# B&R Automation Studio project NewPendant_NG4_11_05_25A
Automation Studio 4.9


## Configuration X20CP1585_MIG_HW_PS

### Task classes (Cpu.sw)
```
Cyclic#1 (cycle 800 us, tolerance 0 us):
  LincolnPS <- Universal.LincolnPS.prg
  Telnet <- Universal.Telnet.prg [disabled]
  TML_srv <- Universal.TML_srv.prg
  AVC_SYNCH <- FourAxisTigCtrl.AVC_SYNCH.prg
Cyclic#2 (cycle 2400 us, tolerance 24000 us):
  TIG_PSprc <- Universal.TIG_PSprc.prg
  WRST <- Universal.WRST.prg
  XMLHelper <- Universal.XMLHelper.prg
  BR_DC <- Universal.BR_DC.prg
  AVCprc <- Universal.AVCprc.prg
  OSC_TMLprc <- Universal.OSC_TMLprc.prg
  WIREprc <- Universal.WIREprc.prg
  HW_PSprc <- Universal.HW_PSprc.prg
  GasCoolPrc <- Universal.GasCoolPrc.prg
  WireBlkPrc <- Universal.WireBlkPrc.prg
  IndexPrc <- Universal.IndexPrc.prg
  TvlRotPrc <- Universal.TvlRotPrc.prg
Cyclic#3 (cycle 51200 us, tolerance 5120000 us):
  MV <- Universal.MV.prg
  HMI_M <- FourAxisTigCtrl.HMI_M.prg
  MiscOper <- Universal.MiscOper.prg
  PermSaving <- FourAxisTigCtrl.PermSaving.prg
  Main2 <- FourAxisTigCtrl.Main2.prg
  DC2DirMtr <- Universal.DC2DirMtr.prg
  TML_RLY <- Universal.TML_RLY.prg
Cyclic#5 (cycle 204800 us, tolerance 204800 us):
  HMI_Report <- FourAxisTigCtrl.HMI_Report.prg
Cyclic#8 (cycle 8000 us, tolerance 40000000 us):
  SuperMstr <- Universal.SuperMstr.prg
  FileOper <- Universal.FileOper.prg
  cJSONTest <- UDP.cJSON.cJSONTest.prg [disabled] (AdditionalLibraryDirectories=\Logical\UDP\sscanf2\, AdditionalLibraries=sscanf2-i386)
  udpserv <- UDP.paiUDPService.udpserv.prg [disabled]
  udpApp <- UDP.udpApp.prg [disabled]
  udpclient <- UDP.paiUDPService.udpclient.prg [disabled]
  udpsimonly <- UDP.udpsimonly.prg [disabled]
DataObjects: Acp10sys, PermObj_15, PermObj_16, PermObj_7, LogBook1, PermObj_3
VcDataObjects: Visu1 <- Visu1.dob, Visu2 <- Visu2.dob, Visu_M <- Visu_M.dob
Binaries: TCData, vccbtn, vcpdvnc, arialbd, vcmgr, vcgclass, vcfile, vccnum, vcfntttf, vcpkat, vcbclass, arial, visvc, vcalarm, vcdsloc, vctcal, vcpfx20, vccshape, vcshared, vcrt, vcnet, vcctext, vcdsint, vcpdsw, vccovl, vcchspot, Visu202, Visu201, udbdef, Visu203, vcpfar00, vcclbox, Visu_M02, vccbmp, Visu_M03, Visu_M01, arialbi, vccstr, vccline, vccddbox, vccpopup, Visu102, Visu101, Visu103, vccdt, Acp10map, acp10cfg, asfw, ashwd, arconfig, iomap, sysconf, ashwac
Libraries: bglibas, asstring, AsXml, sprintf2, AsUDP, Runtime, Acp10man, Acp10par, NcGlobal, sys_lib, brsystem, Library, dvframe, standard, fileio, asiotime, astime, dataobj, powerlnk, astcp, vcresman, visapi, ashw, asbrmath, ashydcon
```

### Hardware
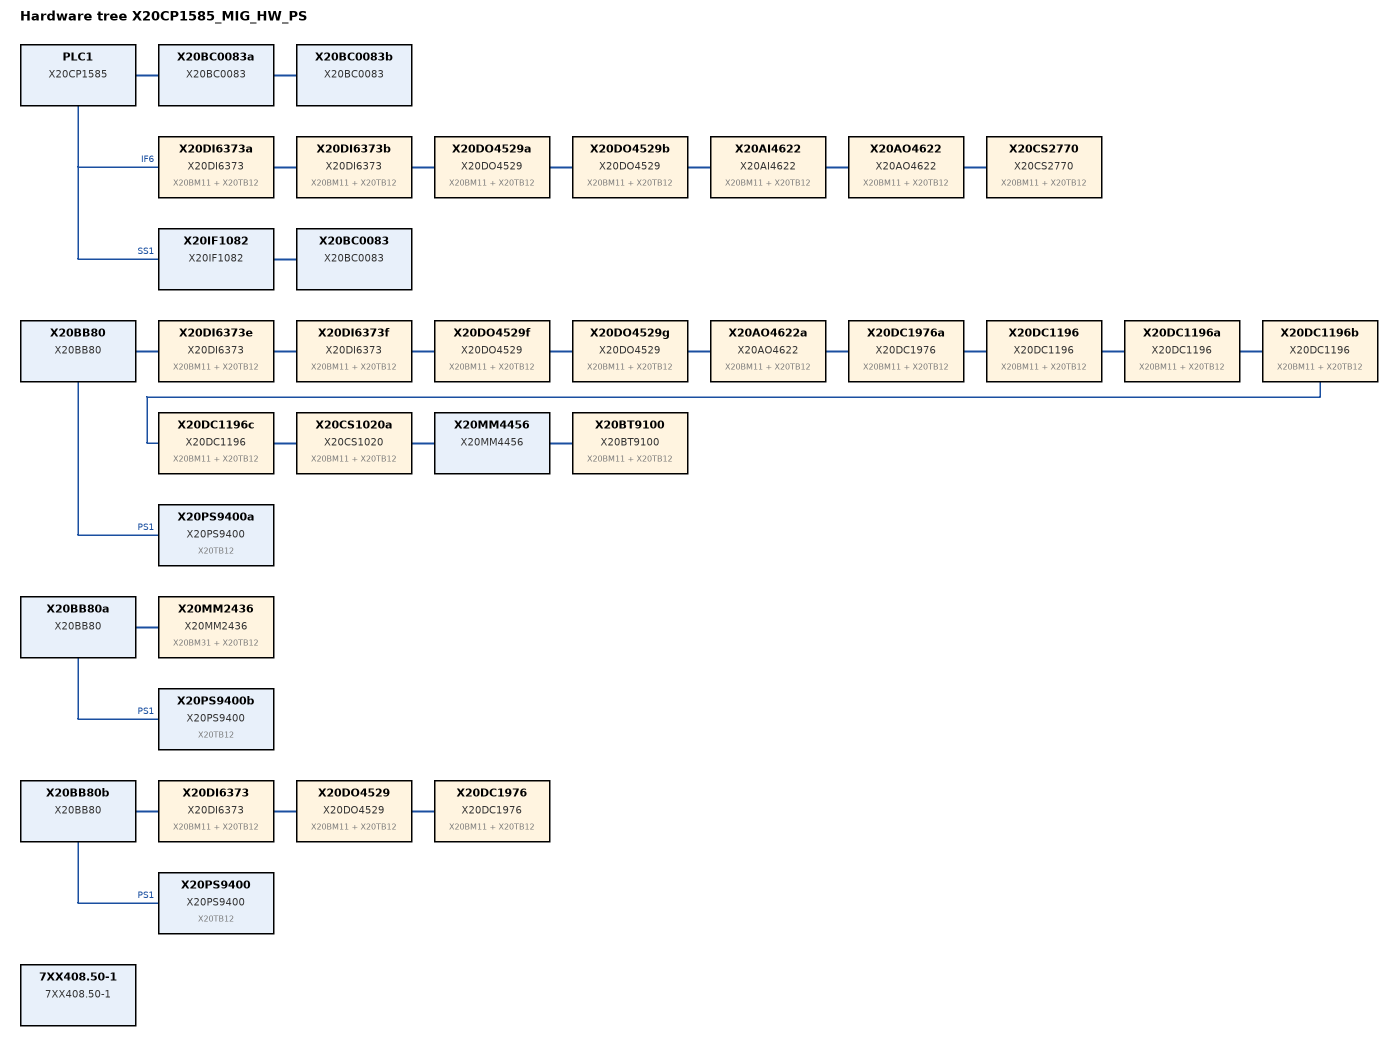
```
7XX408.50-1 : 7XX408.50-1 v1.2.0.0
  Supervision = off
  CounterMode = AB counter
PLC1 : X20CP1585 v1.10.0.0
  Connector IF2:
    ActivateDevice = 1
    Mode = Manual
    InternetAddress = 192.168.10.123
    SubnetMask = 255.255.255.0
    Vnc1
    VncVcObjectName1 = Visu_M
    VncKeyMappingFile1 = VC\PS2-Keyboard.dis
    VncMaxConnections1 = 3
    VncRefreshRate1 = 200
    VncTitle1 = Reports
    Vnc2
    VncVcObjectName2 = Visu2
    VncKeyMappingFile2 = VC\PS2-Keyboard1.dis
    VncPortNumber2 = 5901
    VncMaxConnections2 = 2
    VncRefreshRate2 = 100
    Vnc3
    VncVcObjectName3 = Visu1
    VncKeyMappingFile3 = VC\PS2-Keyboard14.dis
    VncPortNumber3 = 5902
    VncMaxConnections3 = 2
  Connector IF3:
    DNAConfiguration = manual
    CycleTime = 800
    EplNatSubnet = 192.168.102.0
    InaNodeNumber = 1
  Connector IF6:
    CycleTime = 800
  ConfigurationID = UnivCntrl-10-19-21F
  UserPartitionSize = 256
  UserRamSize = 770048
  PermanentPvSize = 96000
  RemanentGlobalPvSize = 15000
  VolatileGlobalPvSize = 3300000
  TimerDeviceType = EPLX2X
  TimerDevice = PLC1.IF3
  TaskClassIdleTime = 1600
  Cyclic1Duration = 800
  Cyclic1Tolerance = 0
  Cyclic1Stack = 16000
  Cyclic2Duration = 2400
  Cyclic2Tolerance = 24000
  Cyclic2Stack = 65536
  Cyclic3Duration = 51200
  Cyclic3Tolerance = 5120000
  Cyclic4Duration = 102400
  Cyclic4Tolerance = 102400
  Cyclic5Duration = 204800
  Cyclic5Tolerance = 204800
  Cyclic6Duration = 409600
  Cyclic6Tolerance = 409600
  Cyclic7Duration = 20000000
  Cyclic7Tolerance = 20000000
  Cyclic8Duration = 8000
  Cyclic8Tolerance = 40000000
  FileDevice1
  FileDeviceName1 = Data
  FileDevicePath1 = f:\Data
  FileDevice2
  FileDeviceName2 = WeldPrograms
  FileDevicePath2 = f:\WeldPrograms
  FileDevice3
  FileDeviceName3 = HMI
  FileDevicePath3 = f:\HMI
  FileDevice4
  FileDeviceName4 = CFG
  FileDevicePath4 = f:\CFG
  FileDevice5
  FileDeviceName5 = TEMP
  FileDevicePath5 = f:\TEMP
  FileDevice6
  FileDeviceName6 = REPORTS
  FileDevicePath6 = f:\Reports
  FtpUser1
  FtpUsername1 = anonymous
  FtpUserPassword1 = ilVrWe+rnGADVB+XCj+0qQ/lTsJeu4vW1xfWuH+9Xv8=
  FtpUserSalt1 = NATz6vdL
  FTPAccessRight1 = 0
X20AI4622 : X20AI4622 v1.2.0.0  [SS1 -> X20TB12c.SS; SL -> X20BM11c.SL1]
  Supervision = off
X20AO4622 : X20AO4622 v1.1.0.0  [SS1 -> X20TB12b.SS; SL -> X20BM11b.SL1]
  Supervision = off
X20AO4622a : X20AO4622 v1.1.0.0 (Disabled=true)  [SS1 -> X20TB12u.SS; SL -> X20BM11q.SL1]
  Supervision = off
X20BB80 : X20BB80 v1.0.2.0 (Disabled=true)
  Connector IF1 (Disabled=true)
    CycleTime = 800
X20BB80a : X20BB80 v1.0.2.0 (Disabled=true)
  Connector IF1 (Disabled=true)
    CycleTime = 800
    BusLength = 1
    Stations = 4
X20BB80b : X20BB80 v1.0.2.0 (Disabled=true)
  Connector IF1 (Disabled=true)
    CycleTime = 800
    AsyncPayload = 120
X20BC0083 : X20BC0083 v2.16.0.0 (Disabled=true)  [PLK1 -> X20IF1082.IF1 (NodeNumber=5) [Cable Type=PowerlinkCable, Length=10, Version=1.0.0.3]; SL -> X20BB80b.SL1]
  Supervision = off
X20BC0083a : X20BC0083 v2.16.0.0 (Disabled=true)  [PLK1 -> PLC1.IF3 (NodeNumber=6) [Cable Type=PowerlinkCable, Length=10, Version=1.0.0.3]; PLK2 -> X20BC0083b.PLK1 (NodeNumber=6) [Cable Type=PowerlinkCable, Length=10, Version=1.0.0.3]; SL -> X20BB80.SL1]
  Supervision = off
X20BC0083b : X20BC0083 v2.16.0.0 (Disabled=true)  [PLK1 -> X20BC0083a.PLK2 (NodeNumber=7) [Cable Type=PowerlinkCable, Length=10, Version=1.0.0.3]; SL -> X20BB80a.SL1]
  Supervision = off
X20BM11 : X20BM11 v1.1.0.0  [X2X1 -> X20BM11e.X2X2]
X20BM11a : X20BM11 v1.1.0.0  [X2X1 -> X20BM11d.X2X2]
X20BM11ab : X20BM11 v1.1.0.0 (Disabled=true)  [X2X1 -> X20BM11z.X2X2]
X20BM11b : X20BM11 v1.1.0.0  [X2X1 -> X20BM11c.X2X2]
X20BM11c : X20BM11 v1.1.0.0  [X2X1 -> X20BM11a.X2X2]
X20BM11d : X20BM11 v1.1.0.0  [X2X1 -> X20BM11.X2X2]
X20BM11e : X20BM11 v1.1.0.0  [X2X1 -> PLC1.IF6]
X20BM11l : X20BM11 v1.1.0.0  [X2X1 -> X20BM11b.X2X2]
X20BM11m : X20BM11 v1.1.0.0 (Disabled=true)  [X2X1 -> X20BB80.IF1]
X20BM11n : X20BM11 v1.1.0.0 (Disabled=true)  [X2X1 -> X20BM11m.X2X2]
X20BM11o : X20BM11 v1.1.0.0 (Disabled=true)  [X2X1 -> X20BM11n.X2X2]
X20BM11p : X20BM11 v1.1.0.0 (Disabled=true)  [X2X1 -> X20BM11o.X2X2]
X20BM11q : X20BM11 v1.1.0.0 (Disabled=true)  [X2X1 -> X20BM11p.X2X2]
X20BM11r : X20BM11 v1.1.0.0 (Disabled=true)  [X2X1 -> X20BM11q.X2X2]
X20BM11s : X20BM11 v1.1.0.0 (Disabled=true)  [X2X1 -> X20BM11r.X2X2]
X20BM11t : X20BM11 v1.1.0.0 (Disabled=true)  [X2X1 -> X20BM11s.X2X2]
X20BM11u : X20BM11 v1.1.0.0 (Disabled=true)  [X2X1 -> X20BM11t.X2X2]
X20BM11v : X20BM11 v1.1.0.0 (Disabled=true)  [X2X1 -> X20BM11u.X2X2]
X20BM11w : X20BM11 v1.1.0.0 (Disabled=true)  [X2X1 -> X20BM11v.X2X2]
X20BM11x : X20BM11 v1.1.0.0 (Disabled=true)  [X2X1 -> X20MM4456.X2X2]
X20BM11y : X20BM11 v1.1.0.0 (Disabled=true)  [X2X1 -> X20BB80b.IF1]
X20BM11z : X20BM11 v1.1.0.0 (Disabled=true)  [X2X1 -> X20BM11y.X2X2]
X20BM31 : X20BM31 v1.1.0.0 (Disabled=true)  [X2X1 -> X20BB80a.IF1]
X20BT9100 : X20BT9100 v1.3.0.0 (Disabled=true)  [SS1 -> X20TB12ab.SS; SL -> X20BM11x.SL1]
  Supervision = off
X20CS1020a : X20CS1020 v1.8.0.0 (Disabled=true)  [SS1 -> X20TB12aa.SS; SL -> X20BM11w.SL1]
  Connector IF1 (Disabled=true)
    ActivateIna = 0
  Supervision = off
X20CS2770 : X20CS2770 v1.9.1.0  [SS1 -> X20TB12n.SS; SL -> X20BM11l.SL1]
  Supervision = off
  CANdataFormat01 = UINT
  Baudrate02 = 250000
  CANdataFormat02 = UINT
X20DC1196 : X20DC1196 v1.4.0.0 (Disabled=true)  [SS1 -> X20TB12w.SS; SL -> X20BM11s.SL1]
  Supervision = off
X20DC1196a : X20DC1196 v1.4.0.0 (Disabled=true)  [SS1 -> X20TB12x.SS; SL -> X20BM11t.SL1]
  Supervision = off
X20DC1196b : X20DC1196 v1.4.0.0 (Disabled=true)  [SS1 -> X20TB12y.SS; SL -> X20BM11u.SL1]
  Supervision = off
X20DC1196c : X20DC1196 v1.4.0.0 (Disabled=true)  [SS1 -> X20TB12z.SS; SL -> X20BM11v.SL1]
  Supervision = off
X20DC1976 : X20DC1976 v1.3.0.0 (Disabled=true)  [SS1 -> X20TB12af.SS; SL -> X20BM11ab.SL1]
  Supervision = off
  BrokenWireConfig = off
X20DC1976a : X20DC1976 v1.3.0.0 (Disabled=true)  [SS1 -> X20TB12v.SS; SL -> X20BM11r.SL1]
  Supervision = off
  BrokenWireConfig = off
X20DI6373 : X20DI6373 v1.0.1.0 (Disabled=true)  [SS1 -> X20TB12ac.SS; SL -> X20BM11y.SL1]
  Supervision = off
X20DI6373a : X20DI6373 v1.0.1.0  [SS1 -> X20TB12e.SS; SL -> X20BM11e.SL1]
  Supervision = off
X20DI6373b : X20DI6373 v1.0.1.0  [SS1 -> X20TB12.SS; SL -> X20BM11.SL1]
  Supervision = off
X20DI6373e : X20DI6373 v1.0.1.0 (Disabled=true)  [SS1 -> X20TB12q.SS; SL -> X20BM11m.SL1]
  Supervision = off
X20DI6373f : X20DI6373 v1.0.1.0 (Disabled=true)  [SS1 -> X20TB12r.SS; SL -> X20BM11n.SL1]
  Supervision = off
X20DO4529 : X20DO4529 v1.2.0.0 (Disabled=true)  [SS1 -> X20TB12ad.SS; SL -> X20BM11z.SL1]
  Supervision = off
X20DO4529a : X20DO4529 v1.2.0.0  [SS1 -> X20TB12d.SS; SL -> X20BM11d.SL1]
  Supervision = off
X20DO4529b : X20DO4529 v1.2.0.0  [SS1 -> X20TB12a.SS; SL -> X20BM11a.SL1]
  Supervision = off
X20DO4529f : X20DO4529 v1.2.0.0 (Disabled=true)  [SS1 -> X20TB12s.SS; SL -> X20BM11o.SL1]
  Supervision = off
X20DO4529g : X20DO4529 v1.2.0.0 (Disabled=true)  [SS1 -> X20TB12t.SS; SL -> X20BM11p.SL1]
  Supervision = off
X20IF1082 : X20IF1082 v1.12.0.0 (Disabled=true)  [SS -> PLC1.SS1]
  Connector IF1 (Disabled=true)
    DNAConfiguration = manual
    CycleTime = 800
    InaNodeNumber = 1
X20MM2436 : X20MM2436 v1.6.0.0 (Disabled=true)  [SS1 -> X20TB12o.SS; SL -> X20BM31.SL1]
  Supervision = off
X20MM4456 : X20MM4456 v1.5.0.0 (Disabled=true)  [X2X1 -> X20BM11w.X2X2]
  Supervision = off
X20PS9400 : X20PS9400 v1.8.0.0 (Disabled=true)  [SS1 -> X20TB12ag.SS; PS -> X20BB80b.PS1]
  Supervision = off
  StatusInfo = off
X20PS9400a : X20PS9400 v1.8.0.0 (Disabled=true)  [SS1 -> X20TB12m.SS; PS -> X20BB80.PS1]
  Supervision = off
X20PS9400b : X20PS9400 v1.8.0.0 (Disabled=true)  [SS1 -> X20TB12p.SS; PS -> X20BB80a.PS1]
  Supervision = off
X20TB12 : X20TB12 v1.0.0.0
X20TB12a : X20TB12 v1.0.0.0
X20TB12aa : X20TB12 v1.0.0.0 (Disabled=true)
X20TB12ab : X20TB12 v1.0.0.0 (Disabled=true)
X20TB12ac : X20TB12 v1.0.0.0 (Disabled=true)
X20TB12ad : X20TB12 v1.0.0.0 (Disabled=true)
X20TB12af : X20TB12 v1.0.0.0 (Disabled=true)
X20TB12ag : X20TB12 v1.0.0.0 (Disabled=true)
X20TB12b : X20TB12 v1.0.0.0
X20TB12c : X20TB12 v1.0.0.0
X20TB12d : X20TB12 v1.0.0.0
X20TB12e : X20TB12 v1.0.0.0
X20TB12m : X20TB12 v1.0.0.0 (Disabled=true)
X20TB12n : X20TB12 v1.0.0.0
X20TB12o : X20TB12 v1.0.0.0 (Disabled=true)
X20TB12p : X20TB12 v1.0.0.0 (Disabled=true)
X20TB12q : X20TB12 v1.0.0.0 (Disabled=true)
X20TB12r : X20TB12 v1.0.0.0 (Disabled=true)
X20TB12s : X20TB12 v1.0.0.0 (Disabled=true)
X20TB12t : X20TB12 v1.0.0.0 (Disabled=true)
X20TB12u : X20TB12 v1.0.0.0 (Disabled=true)
X20TB12v : X20TB12 v1.0.0.0 (Disabled=true)
X20TB12w : X20TB12 v1.0.0.0 (Disabled=true)
X20TB12x : X20TB12 v1.0.0.0 (Disabled=true)
X20TB12y : X20TB12 v1.0.0.0 (Disabled=true)
X20TB12z : X20TB12 v1.0.0.0 (Disabled=true)
```

## Configuration X20CP1685_MIG_HW_PS

CPU X20CP1685, AutomationRuntime J4.93, Build 4.1.2, Safety 1.10, Vc V4.73.1

### IoMap.iom - PLC1/IoMap.iom
```iecst
(********************************************************************
 * COPYRIGHT -- wsi
 ********************************************************************
 * File: IoMap.iom
 * Author: wsi
 * Created: May 14, 2013
 ********************************************************************
 * IO mapping file
 ********************************************************************)
VAR_CONFIG
	::hardware.Inputs[0] AT %IX."X20DI6373e".DigitalInput01;
	::hardware.Inputs[1] AT %IX."X20DI6373e".DigitalInput02;
	::hardware.Inputs[2] AT %IX."X20DI6373e".DigitalInput03;
	::hardware.Inputs[3] AT %IX."X20DI6373e".DigitalInput04;
	::hardware.Inputs[4] AT %IX."X20DI6373e".DigitalInput05;
	::hardware.Inputs[6] AT %IX."X20DI6373f".DigitalInput01;
	::hardware.Inputs[7] AT %IX."X20DI6373f".DigitalInput02;
	::hardware.Inputs[8] AT %IX."X20DI6373f".DigitalInput03;
	::hardware.Inputs[9] AT %IX."X20DI6373f".DigitalInput04 INVERSE;
	Hardware[1].Inp[5] AT %IX."X20DI6373f".DigitalInput05; (*Gas Sensor*)
	Hardware[1].Inp[4] AT %IX."X20DI6373f".DigitalInput06; (*Coolant sensor*)
	::hardware.Inputs[13] AT %IX."X20DC1976a".DigitalInput02;
	::hardware.Inputs[14] AT %IX."X20DC1196".DigitalInput01;
	::hardware.Inputs[15] AT %IX."X20DC1196".DigitalInput02;
	::hardware.Inputs[16] AT %IX."X20DC1196a".DigitalInput01;
	::hardware.Inputs[17] AT %IX."X20DC1196a".DigitalInput02;
	::hardware.Inputs[18] AT %IX."X20DC1196b".DigitalInput01;
	::hardware.Inputs[19] AT %IX."X20DC1196b".DigitalInput02;
	::hardware.Inputs[20] AT %IX."X20DC1196c".DigitalInput01;
	::hardware.Inputs[21] AT %IX."X20DC1196c".DigitalInput02;
	::hardware.Outputs[0] AT %QX."X20DO4529f".DigitalOutput01;
	::hardware.Outputs[1] AT %QX."X20DO4529f".DigitalOutput02;
	::hardware.Outputs[2] AT %QX."X20DO4529f".DigitalOutput03;
	::hardware.Outputs[3] AT %QX."X20DO4529f".DigitalOutput04;
	::hardware.Outputs[4] AT %QX."X20DO4529g".DigitalOutput01;
	::hardware.Outputs[5] AT %QX."X20DO4529g".DigitalOutput02;
	::hardware.Outputs[6] AT %QX."X20DO4529g".DigitalOutput03;
	Hardware[1].Outp[4] AT %QX."X20DO4529g".DigitalOutput04; (*Gas Solenoid*)
	::hardware.AnalogOutputs[0] AT %QW."X20AO4622a".AnalogOutput01;
	::hardware.AnalogOutputs[1] AT %QW."X20AO4622a".AnalogOutput02;
	::hardware.AnalogOutputs[2] AT %QW."X20AO4622a".AnalogOutput03;
	::hardware.AnalogOutputs[3] AT %QW."X20AO4622a".AnalogOutput04;
	::motors[0].Hardware.PeriodDurationPWM AT %QW."X20MM4456".PeriodDurationPWM;
	::motors[0].Hardware.PulseWidthPWM AT %QW."X20MM4456".PulseWidthCurrentPWM01;
	::motors[1].Hardware.PulseWidthPWM AT %QW."X20MM4456".PulseWidthCurrentPWM02;
	::motors[2].Hardware.PulseWidthPWM AT %QW."X20MM4456".PulseWidthCurrentPWM03;
	::motors[3].Hardware.PulseWidthPWM AT %QW."X20MM4456".PulseWidthCurrentPWM04;
	::motors[0].Hardware.Counter AT %IW."X20DC1196".Encoder01;
	::motors[1].Hardware.Counter AT %IW."X20DC1196a".Encoder01;
	::motors[2].Hardware.Counter AT %IW."X20DC1196b".Encoder01;
	::motors[3].Hardware.Counter AT %IW."X20DC1196c".Encoder01;
	::hardware.Inputs[22] AT %IX."X20DI6373".DigitalInput01;
	::hardware.Inputs[23] AT %IX."X20DI6373".DigitalInput02;
	::hardware.Inputs[24] AT %IX."X20DI6373".DigitalInput03;
	::hardware.Inputs[25] AT %IX."X20DI6373".DigitalInput04;
	::hardware.Inputs[26] AT %IX."X20DI6373".DigitalInput05;
	::hardware.Inputs[27] AT %IX."X20DI6373".DigitalInput06;
	::hardware.Outputs[8] AT %QX."X20DO4529".DigitalOutput01;
	::hardware.Outputs[9] AT %QX."X20DO4529".DigitalOutput02;
	::hardware.Outputs[10] AT %QX."X20DO4529".DigitalOutput03;
	::hardware.Outputs[11] AT %QX."X20DO4529".DigitalOutput04;
	::hardware.Inputs[29] AT %IX."X20DC1976".DigitalInput02;
	::menu[1].Counter AT %IW."X20DC1976".Encoder01;
	::menu[1].MenuButton AT %IX."X20DC1976".DigitalInput01;
	::motors[0].Hardware.PWMError AT %IX."X20MM4456".PWMError01;
	::motors[0].Hardware.CurrentError AT %IX."X20MM4456".CurrentError01;
	::motors[0].Hardware.OverCurrentError AT %IX."X20MM4456".OverCurrentError01;
	::hardware.PWM_Status.UnderVoltageError AT %IX."X20MM4456".UnderVoltageError;
	::hardware.PWM_Status.VolatgeWarning AT %IX."X20MM4456".VoltageWarning;
	::hardware.PWM_Status.OverVoltageError AT %IX."X20MM4456".OverVoltageError;
	::hardware.PWM_Status.OvertempeatureError AT %IX."X20MM4456".OvertemperatureError;
	::motors[0].Hardware.ClearError AT %QX."X20MM4456".ResetCounter01;
	::motors[1].Hardware.ClearError AT %QX."X20MM4456".ClearError02;
	::motors[2].Hardware.ClearError AT %QX."X20MM4456".ClearError03;
	::motors[3].Hardware.ClearError AT %QX."X20MM4456".ClearError04;
	::motors[2].Hardware.PWMError AT %IX."X20MM4456".PWMError03;
	::motors[1].Hardware.PWMError AT %IX."X20MM4456".PWMError02;
	::motors[2].Hardware.CurrentError AT %IX."X20MM4456".CurrentError03;
	::motors[3].Hardware.CurrentError AT %IX."X20MM4456".CurrentError04;
	::motors[3].Hardware.PWMError AT %IX."X20MM4456".PWMError04;
	::motors[1].Hardware.OverCurrentError AT %IX."X20MM4456".OverCurrentError02;
	::motors[2].Hardware.OverCurrentError AT %IX."X20MM4456".OverCurrentError03;
	::motors[3].Hardware.OverCurrentError AT %IX."X20MM4456".OverCurrentError04;
	::motors[1].Hardware.CurrentError AT %IX."X20MM4456".CurrentError02;
	::Pendant[0].SerialNumber AT %ID."7XX408.50-1".SerialNumber;
	::Pendant[0].Inp[0] AT %IX."7XX408.50-1".DigitalInput03;
	::Pendant[0].Inp[1] AT %IX."7XX408.50-1".DigitalInput04;
	::Pendant[0].Inp[2] AT %IX."7XX408.50-1".DigitalInput05;
	::Pendant[0].Inp[3] AT %IX."7XX408.50-1".DigitalInput06;
	::Pendant[0].Inp[4] AT %IX."7XX408.50-1".DigitalInput07;
	::Pendant[0].Inp[5] AT %IX."7XX408.50-1".DigitalInput08;
	::Pendant[0].Inp[6] AT %IX."7XX408.50-1".DigitalInput09;
	::Pendant[0].Inp[7] AT %IX."7XX408.50-1".DigitalInput10;
	::Pendant[0].Inp[8] AT %IX."7XX408.50-1".DigitalInput11;
	::Pendant[0].Inp[9] AT %IX."7XX408.50-1".DigitalInput12;
	::Pendant[0].Inp[10] AT %IX."7XX408.50-1".DigitalInput13;
	::Pendant[0].Inp[11] AT %IX."7XX408.50-1".DigitalInput14;
	::Pendant[0].Inp[12] AT %IX."7XX408.50-1".DigitalInput15;
	::Pendant[0].Inp[13] AT %IX."7XX408.50-1".DigitalInput16;
	::Pendant[0].Outp[0] AT %QX."7XX408.50-1".DigitalOutput01;
	::Pendant[0].Outp[1] AT %QX."7XX408.50-1".DigitalOutput02;
	::Pendant[0].Outp[2] AT %QX."7XX408.50-1".DigitalOutput03;
	::Pendant[0].Outp[3] AT %QX."7XX408.50-1".DigitalOutput04;
	::Pendant[0].Outp[4] AT %QX."7XX408.50-1".DigitalOutput05;
	::Pendant[0].Outp[5] AT %QX."7XX408.50-1".DigitalOutput06;
	::Pendant[0].Outp[6] AT %QX."7XX408.50-1".DigitalOutput07;
	::Pendant[0].Outp[7] AT %QX."7XX408.50-1".DigitalOutput08;
	::Pendant[0].Outp[8] AT %QX."7XX408.50-1".DigitalOutput09;
	::Pendant[0].Outp[9] AT %QX."7XX408.50-1".DigitalOutput10;
	::Pendant[0].Outp[10] AT %QX."7XX408.50-1".DigitalOutput11;
	::Pendant[0].Outp[11] AT %QX."7XX408.50-1".DigitalOutput12;
	::Pendant[0].Outp[12] AT %QX."7XX408.50-1".DigitalOutput13;
	::Pendant[0].Outp[13] AT %QX."7XX408.50-1".DigitalOutput14;
	::Pendant[0].Outp[14] AT %QX."7XX408.50-1".DigitalOutput15;
	::Pendant[0].Outp[15] AT %QX."7XX408.50-1".DigitalOutput16;
	::Pendant[0].ABEncoder AT %ID."7XX408.50-1".ABEncoder01;
	::Pendant[0].NotWheelReset AT %QX."7XX408.50-1".NotCounterReset;
	::TML_mgr[0].hrdw[0].RXCount AT %IB."X20CS2770".RX01Count;
	::TML_mgr[0].hrdw[0].TXCountReadBack AT %IB."X20CS2770".TX01CountReadBack;
	::TML_mgr[0].hrdw[0].RXDataSize0 AT %IB."X20CS2770".RX01DataSize;
	::TML_mgr[0].hrdw[0].RXIdent0 AT %ID."X20CS2770".RX01Ident;
	::TML_mgr[0].hrdw[0].RXData0Word0[0] AT %IW."X20CS2770".RX01DataWord0;
	::TML_mgr[0].hrdw[0].RXData0Word0[1] AT %IW."X20CS2770".RX01DataWord1;
	::TML_mgr[0].hrdw[0].RXData0Word0[2] AT %IW."X20CS2770".RX01DataWord2;
	::TML_mgr[0].hrdw[0].RXData0Word0[3] AT %IW."X20CS2770".RX01DataWord3;
	::TML_mgr[0].hrdw[0].TXCount AT %QB."X20CS2770".TX01Count;
	::TML_mgr[0].hrdw[0].TXDataSize AT %QB."X20CS2770".TX01DataSize; (*Data length TX object *)
	::TML_mgr[0].hrdw[0].TXIdent AT %QD."X20CS2770".TX01Ident;
	::TML_mgr[0].hrdw[0].TXDataWord0[0] AT %QW."X20CS2770".TX01DataWord0;
	::TML_mgr[0].hrdw[0].TXDataWord0[1] AT %QW."X20CS2770".TX01DataWord1;
	::TML_mgr[0].hrdw[0].TXDataWord0[2] AT %QW."X20CS2770".TX01DataWord2;
	::TML_mgr[0].hrdw[0].TXDataWord0[3] AT %QW."X20CS2770".TX01DataWord3;
	::TML_mgr[0].hrdw[1].RXCount AT %IB."X20CS2770".RX02Count;
	::TML_mgr[0].hrdw[1].TXCountReadBack AT %IB."X20CS2770".TX02CountReadBack;
	::TML_mgr[0].hrdw[1].RXDataSize0 AT %IB."X20CS2770".RX02DataSize;
	::TML_mgr[0].hrdw[1].RXIdent0 AT %ID."X20CS2770".RX02Ident;
	::TML_mgr[0].hrdw[1].RXData0Word0[0] AT %IW."X20CS2770".RX02DataWord0;
	::TML_mgr[0].hrdw[1].RXData0Word0[1] AT %IW."X20CS2770".RX02DataWord1;
	::TML_mgr[0].hrdw[1].RXData0Word0[2] AT %IW."X20CS2770".RX02DataWord2;
	::TML_mgr[0].hrdw[1].RXData0Word0[3] AT %IW."X20CS2770".RX02DataWord3;
	::TML_mgr[0].hrdw[1].TXCount AT %QB."X20CS2770".TX02Count;
	::TML_mgr[0].hrdw[1].TXDataSize AT %QB."X20CS2770".TX02DataSize; (*Data length TX object *)
	::TML_mgr[0].hrdw[1].TXIdent AT %QD."X20CS2770".TX02Ident;
	::TML_mgr[0].hrdw[1].TXDataWord0[0] AT %QW."X20CS2770".TX02DataWord0;
	::TML_mgr[0].hrdw[1].TXDataWord0[1] AT %QW."X20CS2770".TX02DataWord1;
	::TML_mgr[0].hrdw[1].TXDataWord0[2] AT %QW."X20CS2770".TX02DataWord2;
	::TML_mgr[0].hrdw[1].TXDataWord0[3] AT %QW."X20CS2770".TX02DataWord3;
	::Hardware[2].PWM[0].PulseWidthPWM[0] AT %QW."X20MM2436".PulseWidthCurrentPWM01;
	::Hardware[2].PWM[0].PulseWidthPWM[1] AT %QW."X20MM2436".PulseWidthCurrentPWM02;
	::Hardware[2].PWM[0].PeriodDurationPWM AT %QW."X20MM2436".PeriodDurationPWM01PWM02;
	::Hardware[2].PWM[0].SerialNumber AT %ID."X20MM2436".SerialNumber;
	::Hardware[2].PWM[0].ModuleID AT %IW."X20MM2436".ModuleID;
	::Hardware[2].PWM[0].HardwareVariant AT %IW."X20MM2436".HardwareVariant;
	::Hardware[2].PWM[0].FirmwareVersion AT %IW."X20MM2436".FirmwareVersion;
	::Hardware[2].PWM[0].ClearError[0] AT %QX."X20MM2436".ClearError01;
	::Hardware[2].PWM[0].ClearError[1] AT %QX."X20MM2436".ClearError02;
	::Hardware[2].PWM[0].DitherDisable[0] AT %QX."X20MM2436".DitherDisable01;
	::Hardware[2].PWM[0].DitherDisable[1] AT %QX."X20MM2436".DitherDisable02;
	::Hardware[2].PWM[0].ResetCounter[0] AT %QX."X20MM2436".CounterReset01;
	::Hardware[2].PWM[0].ResetCounter[1] AT %QX."X20MM2436".CounterReset02;
	::Hardware[2].PWM[0].Counter[0] AT %IW."X20MM2436".Counter01;
	::Hardware[2].PWM[0].Counter[1] AT %IW."X20MM2436".Counter02;
	::Hardware[2].PWM[0].UnderVoltageError AT %IX."X20MM2436".UnderVoltageError;
	::Hardware[2].PWM[0].OverVoltageError AT %IX."X20MM2436".OverVoltageError;
	::Hardware[2].PWM[0].OvertempeatureError AT %IX."X20MM2436".OvertemperatureError;
	::Hardware[2].PWM[0].CurrentError[0] AT %IX."X20MM2436".CurrentError01;
	::Hardware[2].PWM[0].CurrentError[1] AT %IX."X20MM2436".CurrentError02;
	::Hardware[2].PWM[0].OverCurrentError[0] AT %IX."X20MM2436".OverCurrentError01;
	::Hardware[2].PWM[0].OverCurrentError[1] AT %IX."X20MM2436".OverCurrentError02;
	::Hardware[1].CouplerOK[0] AT %IX."X20BC0083a".ModuleOk;
	::hardware.Inputs[5] AT %IX."X20DI6373a".DigitalInput06;
	Hardware[1].Outp[7] AT %QX."X20DO4529a".DigitalOutput04;
	::Main2:TIG_MIG_Sw_Inp AT %IX."X20DI6373a".DigitalInput03;
	::Hardware[1].Outp[4] AT %QX."X20DO4529b".DigitalOutput02;
	Hardware[1].Outp[2] AT %QX."X20DO4529a".DigitalOutput03;
	Hardware[1].Anal_Outp[0] AT %QW."X20AO4622".AnalogOutput01;
	::Main2:MIG_ESTOP_Rst_Btn_Inp AT %IX."X20DI6373b".DigitalInput06;
	::Main2:MIG_ESTOP_Rst_Out AT %QX."X20DO4529b".DigitalOutput01;
	::Main2:MIG_Btn_Stop_Inp AT %IX."X20DI6373b".DigitalInput01;
	::Main2:MIG_Btn_Right_Inp AT %IX."X20DI6373b".DigitalInput04;
	::Main2:MIG_Btn_Left_Inp AT %IX."X20DI6373b".DigitalInput05;
END_VAR
```

## Configuration test

### Task classes (Cpu.sw)
```
Cyclic#3:
  CK_test <- CK_test.prg
Binaries: gcloader, sysconf, iomap, arconfig, asfw
```

## Logical view

Binary libraries used (declarations not repeated): Acp10man 3.18.2, asstring, AsTCP

- .gitignore (not shown)

### Program Logical/bglib

#### bgBufMemAlloc.h
```c
/**\file: bgBufMemAlloc.h
*Buffer memory (user supplied memory) simple allocation methods.
*/
#ifndef _BG_BUFMEMALLOC_H
#define _BG_BUFMEMALLOC_H

/**
\def BGBUFMEMALLOC_MAX_BLOCKS
Defines maximum number of items within the list of memory blocks.
Used for data object: \link bgBufMemAlloc_typ \endlink
*/
#define BGBUFMEMALLOC_MAX_BLOCKS	16

/**
\struct bgBufMemAlloc_typ
Data object that holds information about simple memory allocation method.\n
In a deeply embedded systems, memory allocation is rather uncommon practice. However,
there are situations (i.e. networking) where certain, simplified "mem allocation" scheme
is rather useful.\n
This data object and associated methods implement memory allocation scheme that uses
user suppllied memory buffer as the "source memory".
*/
typedef struct bgBufMemAlloc_typ{
	char* pBufMem;			/**<Input: User supplied memory buffer*/
	int lengthBufMemBytes; 	/**<Input: Lenght (bytes) of the user supplied memory buffer*/

    int countMaxBlocks;		/**<Input(const): Max number of mem blocks*/
    int countUsedBlocks;	/**<Output: Number of currently allocated blocks*/
    int lengthUsedMemBytes;	/**<Output: Total length (bytes) of currently allocated memory*/

    struct bgBufMemBlock_typ{
		int 	used;			/**<I/O: 0-block not used; 1-block is used*/
        char*   pMemBlock;		/**<Output: Ptr to the mem block*/
        int     lengthMemBlockBytes;	/**<Input: Size (bytes) of the mem block*/
    }memBlock[BGBUFMEMALLOC_MAX_BLOCKS];

}bgBufMemAlloc_typ;

/**
Init method for data object: \link bgBufMemAlloc_typ \endlink
\param p Ptr to data object: \link bgBufMemAlloc_typ \endlink
\param pBufMem Ptr to user supplied memory buffer
\param lengthBufMemBytes Size of the user supplied memory buffer
<b>IMPORTANT: </b>This method <b>must be always</b> called first for the associated data object!\n

*/
void bgBufMemAllocInit(bgBufMemAlloc_typ* p, char* pBufMem, int lengthBufMemBytes);

/**
Method for data object: \link bgBufMemAlloc_typ \endlink\n
Creates / allocates memory block of size (sizeMemBlock)
\param p Ptr to data object: \link bgBufMemAlloc_typ \endlink
\param blockSize Requested memory block size
\param pMemBlock Address to store the pointer to newly allocated mem block
\param sizeMemBlock Address to store the size of the newly allocated mem block
\return Id for the allocated mem block (0 to (BGBUFMEMALLOC_MAX_BLOCKS-1))
*/
int bgBufMemAllocCreateBlock(bgBufMemAlloc_typ* p, int blockSize, char** pMemBlock, int* sizeMemBlock);

/**
Method for data object: \link bgBufMemAlloc_typ \endlink\n
Give the memblock Id, returns the memory and size of the requesed memblock
\param p Ptr to data object: \link bgBufMemAlloc_typ \endlink
\param blockId Id of the mem block previosly allocated using \link bgBufMemAllocCreateBlock \endlink
\param blockSize Address to store the size of the newly allocated mem block
\return Address of the newly allocated mem block or NULL (in case the blockId is invalid)
*/
char* bgBufMemAllocGetBlockPtr(bgBufMemAlloc_typ* p, int blockId, int* blockSize);

/*
##################################################################################
String heap
##################################################################################
*/

/**
\struct bgStringHeap_typ
Data object that holds information about simple memory allocation method for strings.\n
In a deeply embedded systems, dynamic string memory allocation is rather uncommon practice.
However, there are situations (i.e. networking) where certain, simplified dynamic allocation
scheme for storing variable lenght strings is rather useful.\n
This data object and associated methods implement dynamic memory allocation scheme for
strings that uses user suppllied memory buffer as a memory to store variable length strings.
*/
typedef struct bgStringHeap_typ{
	char* pMemStart;	/**<Start of the user supplied memory buffer*/
	int	memSize;		/**<Size (bytes) of the user supplied memory buffer*/
	char* pMemCurrent;	/**<Ptr to the current free memory location within the (pMemStart)*/
	int memFree;		/**<Size (bytes) of still available / free memory*/
}bgStringHeap_typ;

/**
Method for data object: \link bgStringHeap_typ \endlink\n
Creates / allocates memory block of size (sizeMemBlock)
\param pHeap Ptr to data object: \link bgStringHeap_typ \endlink
\param pHeapMem User supplied memory that will be used for storage of dynamic strings
\param memSize Size of the user supplied memory
\return Ptr to the start of memory (same as pHeapMem) or NULL if error
<b>IMPORTANT: </b>This method <b>must be always</b> called first for the associated data object!\n
*/
char* bgStringHeapInit(bgStringHeap_typ* pHeap, char* pHeapMem, int memSize);

/**
Method for data object: \link bgStringHeap_typ \endlink\n
Stores given string (pStr) to the string heap memory. Returns ptr to the stored string.
\param pHeap Ptr to data object: \link bgStringHeap_typ \endlink
\param pStr String to store on the string heap
\return Ptr to string stored on the heap or NULL if error (not enough space)
*/
char* bgStringHeapAddString(bgStringHeap_typ* pHeap, char* pStr);

#endif
```

#### bgdebug.h
```c
#ifndef _BG_DEBUG_H
#define _BG_DEBUG_H

#ifdef WIN32
#define DBG printf
#define DBGMSG printf

#define DBGCRT printf
#define DBGERR printf
#define DBGWAR printf
#define DBGINF printf
#define DBGDBG printf

#else

#include <bur/plc.h>
#include "bgsprintf.h"
#include "bgringbuffer.h"

#define BG_DEBUG_LEVEL_CRITICAL		0
#define BG_DEBUG_LEVEL_ERROR		1
#define BG_DEBUG_LEVEL_WARNING		2
#define BG_DEBUG_LEVEL_INFO			3
#define BG_DEBUG_LEVEL_DEBUG		4

#define BG_DEBUG_UNUSED	0x0

/*
- To completly remove debug msgs from the source code use:
#define BG_DEBUG_ENABLE 0
*/
#define BG_DEBUG_ENABLE 1

/*ptr to global ring buffer for debug messages*/
_GLOBAL bgRingBuffer_typ gRingBuffer;

#if BG_DEBUG_ENABLE == 1
/*BG_DEBUG_ENABLE == 1 => debug messages present in the source code*/
#define DBG(format, args...)	bgRingBuffPutDbgInfo(&gRingBuffer, __FILE__, __FUNCTION__, BG_DEBUG_LEVEL_CRITICAL, BG_DEBUG_UNUSED, format, ## args);
#define DBGMSG(format, args...)	bgRingBuffPrintf(&gRingBuffer, format, ## args);

#define DBGCRT(format, args...)	bgRingBuffPutDbgInfo(&gRingBuffer, __FILE__, __FUNCTION__, BG_DEBUG_LEVEL_CRITICAL, BG_DEBUG_UNUSED, format, ## args);
#define DBGERR(format, args...)	bgRingBuffPutDbgInfo(&gRingBuffer, __FILE__, __FUNCTION__, BG_DEBUG_LEVEL_ERROR, BG_DEBUG_UNUSED, format, ## args);
#define DBGWAR(format, args...)	bgRingBuffPutDbgInfo(&gRingBuffer, __FILE__, __FUNCTION__, BG_DEBUG_LEVEL_WARNING, BG_DEBUG_UNUSED, format, ## args);
#define DBGINF(format, args...)	bgRingBuffPutDbgInfo(&gRingBuffer, __FILE__, __FUNCTION__, BG_DEBUG_LEVEL_INFO, BG_DEBUG_UNUSED, format, ## args);
#define DBGDBG(format, args...)	bgRingBuffPutDbgInfo(&gRingBuffer, __FILE__, __FUNCTION__, BG_DEBUG_LEVEL_DEBUG, BG_DEBUG_UNUSED, format, ## args);

#else
/*BG_DEBUG_ENABLE == 0 => all debug messages removed from the source code*/
#define DBG(format, args...)  ;
#define DBGMSG(format, args...)  ;

#define DBGCRT(format, args...)	;
#define DBGERR(format, args...)	;
#define DBGWAR(format, args...)	;
#define DBGINF(format, args...)	;
#define DBGDBG(format, args...)	;

#endif /*#if BG_DEBUG_ENABLE*/

#endif /*#ifdef WIN32*/

#endif /*#ifndef _BG_DEBUG_H*/
```

#### bgfsig.c
```c
#include <bur/plc.h>
#include <bur/plctypes.h>

#include "bglib/bgdebug.h"
#include "bglib/bgstring.h"
#include "bglib/bgSecMD5Signature.h"
#include "bgfsig.h"

/*define a limit for number of lines within a file*/
#define MAX_NUMBER_OF_LINES	3000

static int bgGetLineFromTextBuffer(char* pText, char** pLineNext, char* pDest, int maxLen, int* charCount);

#define  secretWord "NONE!"

/*=============================================================*/
int bgFileSignatureVerify(char *inFileBuffer, char *resultStringMinLen64)
{
int i, index;
char lineBuffer[255];
char lineBufferRaw[255];
int lineCount;
int charCount;
bgStringList_typ splitLine;
md5_state_t state;
md5_byte_t digest[16];
char hexDigestCalculated[40];
char hexDigestFromFile[40];

char *pLineCurrent;
char *pLineNext;

	/*init digest*/
	md5_init(&state);

	/*init hexDigestFromFile as empty*/
	hexDigestFromFile[0] = 0;

	/*init line ptr-s*/
	pLineCurrent = inFileBuffer;
	pLineNext = 0L;

	lineCount = 0;

	/*process all lines from the file*/
	while( 1 ){
	int isNextLinePresent;

		isNextLinePresent = bgGetLineFromTextBuffer(pLineCurrent, &pLineNext, lineBufferRaw, 255, &charCount);

		if( lineCount++ > MAX_NUMBER_OF_LINES){
			DBGCRT("Supplied file buffer has more then %d lines!\r\n", lineCount);
			if( resultStringMinLen64 )
				strcpy(resultStringMinLen64, "Err: file is too long!");
			return -2;
		}

		/*copy a trimmed line into the local buffer*/
		charCount = bgStrCpyNTrimLeadingSpaces(lineBuffer, lineBufferRaw, 255);

		/*check for empty lines & comments*/
		if( !charCount || (lineBuffer[0] == '*')){
			/*empty lines or comments -> skip and go to the next line*/
		}else{
			/*check if this is a signature line*/
			index = bgStrFind(lineBuffer, "SIGNATURE", -1, 0);
			if( index >= 0){
				/*line w. signature -> extract signature stored in the file*/
				splitLine.src = lineBuffer;
				bgStringSplitLine(&splitLine, '=');
				if( splitLine.itemCount != 2){
					DBGCRT("Can't extract signature from the supplied file buffer\r\n");
					if( resultStringMinLen64 )
						strcpy(resultStringMinLen64, "Err: can't extract signature");
					return -2;
				}
				/*copy extracted signature from the file into the local buffer*/
				bgStrCpyN(hexDigestFromFile, splitLine.items[1], 40);
				bgStringUpper(hexDigestFromFile);

			}else{
				/*line wo. signature -> use (append) for digest calculation*/
				md5_append(&state, (const md5_byte_t *)lineBuffer, strlen(lineBuffer));
			}
		}

		/*process next line*/
		if( isNextLinePresent )
			pLineCurrent = pLineNext;
		else
			break;
	}

	/*append secret content*/
	md5_append(&state, (const md5_byte_t *)secretWord, strlen(secretWord));

	/*generate digest*/
	md5_finish(&state, digest);

	/*convert calculated digest into a hex string*/
	for (i = 0; i < 16; ++i)
	    bgsprintf(hexDigestCalculated + i * 2, "%02X", digest[i]);

	/*check if supplied file buffer had stored digital signature*/
	if( !hexDigestFromFile[0] ){
		/*digital signature was NOT present in this file->return result and current (calculated) file digest*/
		if( resultStringMinLen64 )
			bgsprintf(resultStringMinLen64, "StoredSig=NONE CalcSig=%s\n\r", hexDigestCalculated);
		return 0;

	}else{
		/*digital signature IS present in this file->compare calculated and stored signaure*/

		for (i = 0; i < 32; i++){
			if(hexDigestCalculated[i] != hexDigestFromFile[i] ){
				/*digital signatures are not equal -> exit*/
				if( resultStringMinLen64 )
					bgsprintf(resultStringMinLen64, "StoredSig=%s CalcSig=%s\n\r", hexDigestFromFile, hexDigestCalculated);

				return 2;
			}
		}

		/*digital signature verified! stored and calculated signatures are equal!*/
		if( resultStringMinLen64 )
			bgsprintf(resultStringMinLen64, "StoredSigEQUALCalcSig=%s\n\r", hexDigestCalculated);

		return 1;

	}
}
/*=============================================================*/

/*
Input(s):
char *pText - ptr to the text buffer from which to extract a line
char *pDest - destination buffer where to copy the content of a line
int maxLen - max length of the destination buffer

Output(s):
char **pLineNext - ptr to the next line
int *charCount - total number of chars copied into the dest buffer

Return:
0 - there is no more lines in the supplied text buffer
1 - more lines are present in the supplied text buffer
*/
static int bgGetLineFromTextBuffer(char* pText, char** pLineNext, char* pDest, int maxLen, int* charCount)
{

unsigned char *ptrItemStart, *ptrItemEnd;
unsigned char *ptrCpyDest;

	/*init ptrs to the start of the text buffer*/
	ptrItemStart = pText;
	ptrItemEnd = pText;
	ptrCpyDest = pDest;

	/*basic check*/
	if( *ptrItemStart == 0){
		return 0;
	}

	*charCount = 0;
	while( 1 ){
		if( (*ptrItemEnd == 0x0D) || (*ptrItemEnd == 0x0A)){
			/*EOF line char found! -> exit*/
			ptrItemEnd++;

			/*check for an additional \r or \n*/
			if( (*ptrItemEnd == 0x0D) || (*ptrItemEnd == 0x0A)){
				ptrItemEnd++;
			}

			ptrItemStart = ptrItemEnd;

			/*terminate dest buffer*/
			*ptrCpyDest = 0;

			/*check for an end of the text*/
			if( (*ptrItemEnd == 0) ){
				*pLineNext = 0L;
				/*0 -> there are NO more lines in the text buffer*/
				return 0;
			}else{
				*pLineNext = ptrItemStart;
				/*1 -> there are more lines in the text buffer*/
				return 1;
			}
		}else
		if( *ptrItemEnd == 0){
			/*end of text buffer found! -> exit*/

			/*terminate dest buffer*/
			*ptrCpyDest = 0;

			*pLineNext = 0L;
			/*0 -> there are NO more lines in the text buffer*/
			return 0;
		}else{
			/*copy line content into the supplied dest buffer
			check for buffer overflow*/

			if( (*charCount) < maxLen ){
				*ptrCpyDest = *ptrItemEnd;
				ptrCpyDest++;
				(*charCount)++;
			}else{

				DBGCRT("Line is longer then the max allowed size!\r\n");

				/*terminate dest buffer*/
				*ptrCpyDest = 0;

				*pLineNext = 0L;
				/*0 -> there are NO more lines in the text buffer! Error*/
				return 0;
			}

			ptrItemEnd++;
		}
	}/*while*/
}
```

#### bgstring.c
```c
#ifndef _BG_STRING_C
#define _BG_STRING_C

#ifdef WIN32
#include "string.h"
#else
#include <bur/plctypes.h>
#endif
#include "bgstring.h"

/*
File:
bgString.c

About:
------
- implements  additional string manipulation functions

B&R System Dependencies:
------------------------
- B&R system library: libasstring.a
- B&R system header files: asstring.h

History:
--------
09/11/2005
- rectified issue with bgStringListLines() to properly handle zero length
input string

05/08/2005
-first version

Test and example code:
----------------------
- to run this file standalone:
--- enable following code section (remove or comment out #if 0 / #endif)
--- create cyclic object (task) from C Language and add this file
*/

#if 0
#include <bur/plc.h>
#include <bur/plctypes.h>

#define TXT_SIZE 64
_LOCAL char textBuffer1[TXT_SIZE];
_LOCAL char textBuffer2[TXT_SIZE];
_LOCAL int idxResult;
_LOCAL int idxStart;
_LOCAL int idxEnd;

_INIT void Init(void) {

	/*use defaults*/
	idxStart 	= -1;
	idxEnd 		= -1;
	/*start with empty strings*/
	textBuffer1[0] = 0;
	textBuffer2[0] = 0;
}

_CYCLIC void Cyclic(void) {

	idxResult = bgStrFind(textBuffer1, textBuffer2, start, end);

}
#endif

/*End: Example/Test code*/
int bgStrFind(char *s, char *sub, int idxStart, int idxEnd)
{
	int i, j;
	int subLen;
	char *ptrStr;
	char *ptrSub;

	/*exit if null ptrs*/
	if(!s || !sub)
		return -1;

	/*exit if zero strings*/
	if( !(*s) || !(*sub) )
		return -1;

	subLen = strlen(sub);

	/*check starting index: default = -1 -> start @ s[0]*/
	if(idxStart < 0)
		idxStart = 0;

	/*check end index: default = -1 -> end is sLength - subLength*/
	if(idxEnd < 0){
		idxEnd = strlen(s) - subLen;
	}

	/*check if start is beyond the end*/
	if(idxStart > idxEnd)
		return -1;

	/*search for string <sub> within the string <s>*/
	for(i=idxStart; i<=idxEnd; i++)
	{
		ptrStr = s + i;
		ptrSub = sub;

		for(j=0; j<subLen; j++, ptrStr++, ptrSub++)
		{
			if( *ptrStr!= *ptrSub)
				break;
		}

		if( j == subLen)
			return i;
	}

	return -1;
}

/*
bgStrFindEx - has an extra option
option = 0; same as bgStrFind
option = 1; before comparing, both strings are converted to lower case
*/
int bgStrFindEx(char *s, char *sub, int idxStart, int idxEnd, int option)
{
	int i, j;
	int subLen;
	char *ptrStr;
	char *ptrSub;

	/*exit if null ptrs*/
	if(!s || !sub)
		return -1;

	/*exit if zero strings*/
	if( !(*s) || !(*sub) )
		return -1;

	subLen = strlen(sub);

	/*check starting index: default = -1 -> start @ s[0]*/
	if(idxStart < 0)
		idxStart = 0;

	/*check end index: default = -1 -> end is sLength - subLength*/
	if(idxEnd < 0){
		idxEnd = strlen(s) - subLen;
	}

	/*check if start is beyond the end*/
	if(idxStart > idxEnd)
		return -1;

	/*search for string <sub> within the string <s>*/
	for(i=idxStart; i<=idxEnd; i++)
	{
		ptrStr = s + i;
		ptrSub = sub;

		for(j=0; j<subLen; j++, ptrStr++, ptrSub++)
		{
			if(!option){
				if( *ptrStr!= *ptrSub)
					break;
			}else{
				if( bgCharToLowerCase(*ptrStr) != bgCharToLowerCase(*ptrSub) )
					break;
			}
		}

		if( j == subLen)
			return i;
	}

	return -1;
}

int bgStrCpyN(char *dest, char *src, int maxNoOfCharsToCopy)
{
int i;

	/*maxNoOfCharsToCopy-1 - takes into consideration that supplied max
	length is usually the buffer size, 1 char is needed for null termination
	*/
	for(i=0; i<(maxNoOfCharsToCopy-1);i++){
		*(dest+i)=*(src+i);
		if(! (*(src+i) ) )
			break;
	}

	/*if max reached, terminate dest string*/
	if(i >= (maxNoOfCharsToCopy-1))
		*(dest+i)=0;

	/*string termination is not included in the string length*/
	return i;
}

int bgStrTrimCRLF(char *s)
{
int i;
char c;

	for(i=0;i<255;i++){

		c = s[i];

		if( !c )
			break;

		if( (c == 0xa) || (c == 0xd) ){
			s[i] = 0;
			break;
		}
	}

	return i;
}

int bgStrCpyNTrimLeadingSpaces(char *dest, char *src, int maxNoOfCharsToCopy)
{
int i;
int found;
char *srcStart;

	/*look for leading spaces*/
	found = 0;
	for(i=0; i<(maxNoOfCharsToCopy-1);i++){
		if( *(src+i) != ' ' ){
			srcStart = src + i;
			found = 1;
			break;
		}
	}

	if(!found){
	/*src string is all spaces->set destination to empty string*/
		*dest = 0;
		return 0;
	}

	return bgStrCpyN(dest, srcStart, maxNoOfCharsToCopy);
}

/*
copy string, don't go over the size of dest buffer, trim leading / trailing spaces / convert
to lower case
*/
int bgStrCpyNTrimSpcsToLwr(char *dest, char *src, int maxNoOfCharsToCopy)
{
int i;
char* srcStart = src;
char* srcEnd;
int len = strlen(src);

	if( !len )
		return len;

	/*find src start, avoid leading spaces*/
	while(1){
		if( *srcStart != ' ')
			break;

		if( *srcStart == 0)
			return 0;

		srcStart++;
	}

	/*find src end, trim trailing spaces*/
	srcEnd = (char*)(src + len - 1);
	while(1){
		if( *srcEnd != ' ')
			break;

		if( *srcEnd == 0)
			return 0;

		srcEnd--;
	}

	srcEnd++;

	if( srcStart >= srcEnd )
		return 0;

	for(i=0; i<(maxNoOfCharsToCopy-1); i++){
		dest[i] = bgCharToLowerCase(*srcStart);
		srcStart++;
		if(srcStart >= srcEnd){
			i++;
			break;
		}
	}

	dest[i] = 0;
	return i;
}

int bgIsDigit(char c){
	return ((c>='0') && (c<='9')) ? 1 : 0;
}

#if 0
/*
Test for: bgStringListLinesEx()

The xxxxEx functions use externaly supplied buffer space to store result pointers to
lines / words.
Based on the supplied buffer size, functions will calculate max. number of items (char ptr-s)
that may be stored within the given / allocated storage area.
See: pList->itemCountMax

To test it out, create a new cyclic task then use following code!
*/
#include <bur/plc.h>
#include <bur/plctypes.h>

#include "bglib/bgString.h"
#include "bglib/bgString.c"

#include "bglib/bgdebug.h"
#include "bglib/bgringbuffer.c"

_LOCAL bgStringListEx_typ listLines;
_LOCAL bgStringListEx_typ listWords;
_LOCAL char multiLineTextBuffer[256];
_LOCAL int lineCount;
_LOCAL int wordCount;
_LOCAL int test;
_LOCAL char listPtrBuf[128];    /*this is a "free" storage for list ptr-s! use it with caution!*/

_INIT void init()
{
	strcpy(multiLineTextBuffer, "hello world\r\nThis is a test for second line!\r\nThird line is here and there...\r\nLine #4 : right.left dot !\r\n");
	test = 0;
}

_CYCLIC void cyclic()
{
int i, j;

/*
This is just an example on how to use external / user supplied buffer in order to
store line / word lists. Based on the supplied buffer size, functions will calculate
max. number of items that may be stored within the given / allocated storage area.
See: pList->itemCountMax
*/
char* lineListStorage = &listPtrBuf[0];
char* wordListStorage = &listPtrBuf[64];

	if( test ){
		test = 0;

		lineCount = bgStringListLinesEx(&listLines, multiLineTextBuffer, lineListStorage, 64);
		DBG("multiLineTextBuffer has lineCount=%d lines. (same as listLines.itemCount= %d). Lines are:\r\n", lineCount, listLines.itemCount);
		for(i=0; i<listLines.itemCount; i++){
			DBG("Line[%d]->%s\r\n", i, listLines.items[i]);
			wordCount = bgStringSplitLineEx(&listWords, ' ', listLines.items[i], wordListStorage, 64);
				DBG("     Line[%d] has wordCount=%d words. (same as listWords.itemCount= %d). Words are:\r\n", i, wordCount, listWords.itemCount)
			for(j = 0; j<listWords.itemCount; j++)
				DBG("     Word[%d]->%s\r\n", j, listWords.items[j]);
		}
	}
}
#endif
int bgStringListLines(bgStringList_typ * p){
unsigned char *ptrItemStart, *ptrItemEnd;
int	calcItemCount;

/*
	length = strlen( p->src );
*/
	p->itemCount = 0;

	ptrItemStart = p->src;
	ptrItemEnd = p->src;

	if( *ptrItemStart == 0){
		return 0;
	}

/*process the rest; build list of item pointers*/
	calcItemCount 	= 0;
	while( 1 ){
		if( (*ptrItemEnd == 0x0D) || (*ptrItemEnd == 0x0A)){
			*ptrItemEnd = 0;
			p->items[calcItemCount] = ptrItemStart;
			ptrItemEnd++;

			/*check for an additional \r or \n*/
			if( (*ptrItemEnd == 0x0D) || (*ptrItemEnd == 0x0A)){
				ptrItemEnd++;
			}

			ptrItemStart = ptrItemEnd;
			calcItemCount++;

			if(calcItemCount >= BG_STRINGLIST_MAXITEMCOUNT){
				p->itemCount = calcItemCount;
				return -1;
			}

			/*check for an end of the src string*/
			if( (*ptrItemEnd == 0) ){
				p->itemCount = calcItemCount;
				return calcItemCount;
			}
		}else
		if( *ptrItemEnd == 0){
			p->items[calcItemCount] = ptrItemStart;
			calcItemCount++;
			break;
		}else
			ptrItemEnd++;
	}/*while*/

	p->itemCount = calcItemCount;
	return calcItemCount;
}

void bgStringListExMemSet(bgStringListEx_typ *p, char* pAddrListBuffer, int sizeListBuffer)
{
	/*NOTE: we are going to use supplied char buffer as the storage for the array of char ptr-s!*/
    p->items = (unsigned char**)pAddrListBuffer;

	p->itemCountMax = sizeListBuffer / sizeof(char*);
}

int bgStringListLinesEx(bgStringListEx_typ * p, char* pContentBuffer, char* pAddrListBuffer, int sizeListBuffer){
unsigned char *ptrItemStart, *ptrItemEnd;
int	calcItemCount;

    p->src = (unsigned char*)pContentBuffer;

    /*if mem data is defined, use it; otherwise, mem shall have been set using a separate call to xxxExMemSet()*/
    if(pAddrListBuffer && sizeListBuffer)
        bgStringListExMemSet(p, pAddrListBuffer, sizeListBuffer);

	p->itemCount = 0;

	ptrItemStart = p->src;
	ptrItemEnd = p->src;

	if( *ptrItemStart == 0){
		return 0;
	}

/*process the rest; build list of item pointers*/
	calcItemCount 	= 0;
	while( 1 ){
		if( (*ptrItemEnd == 0x0D) || (*ptrItemEnd == 0x0A)){
			*ptrItemEnd = 0;
			p->items[calcItemCount] = ptrItemStart;
			ptrItemEnd++;

			/*check for an additional \r or \n*/
			if( (*ptrItemEnd == 0x0D) || (*ptrItemEnd == 0x0A)){
				ptrItemEnd++;
			}

			ptrItemStart = ptrItemEnd;
			calcItemCount++;

			if(calcItemCount >= p->itemCountMax){
				p->itemCount = calcItemCount;
				return -1;
			}

			/*check for an end of the src string*/
			if( (*ptrItemEnd == 0) ){
				p->itemCount = calcItemCount;
				return calcItemCount;
			}
		}else
		if( *ptrItemEnd == 0){
			p->items[calcItemCount] = ptrItemStart;
			calcItemCount++;
			break;
		}else
			ptrItemEnd++;
	}/*while*/

	p->itemCount = calcItemCount;
	return calcItemCount;
}

#if 0
Example:
(AS: Make a "C" task; add <filename>.c to the task; copy & paste this code)
#######
#include <bur/plc.h>
#include <bur/plctypes.h>

#include "bgString.h"
#include "bgString.c"

#include "bgdebug.h"

_LOCAL bgStringList_typ myList;
_LOCAL bgStringList_typ mySplitList;
_LOCAL char buffer[256];
_LOCAL int lineCount;
_LOCAL int test;

_INIT void init()
{
	strcpy(buffer, "hello world\r\nwhat is new?\r\nthird line\r\nline #4\r\n");
	test = 0;
}

_CYCLIC void cyclic()
{
int i, j;

	if( test ){
		test = 0;
		myList.src = buffer;
		lineCount = bgStringListLines(&myList);

		for(i=0; i<myList.itemCount; i++){
			DBG("Line[%d]->%s\r\n", i, myList.items[i]);

			mySplitList.src = myList.items[i];
			lineCount = bgStringSplitLine(&mySplitList, ' ');
			for(j = 0; j<mySplitList.itemCount; j++)
				DBG("     Word[%d]->%s\r\n", j, mySplitList.items[j]);
		}
	}
}
######
The above code generates following output (debug telnet client):
>Line[0]->hello world
     Word[0]->hello
     Word[1]->world
Line[1]->what is new?
     Word[0]->what
     Word[1]->is
     Word[2]->new?
Line[2]->third line
     Word[0]->third
     Word[1]->line
Line[3]->line #4
     Word[0]->line
     Word[1]->#4

#endif
int bgStringSplitLine(bgStringList_typ * p, char separator){
unsigned char *ptrItemStart, *ptrItemEnd;
int	calcItemCount;

	p->itemCount = 0;

	ptrItemStart = p->src;
	ptrItemEnd = p->src;

/*process the rest; build list of item pointers*/
	calcItemCount 	= 0;
	while( 1 ){
		if( (*ptrItemEnd == separator) ){
			*ptrItemEnd = 0;
			p->items[calcItemCount] = ptrItemStart;
			ptrItemEnd++;

			calcItemCount++;

			/*check for an additional separtor */
			while( (*ptrItemEnd == separator) ){
				ptrItemEnd++;
				if( (*ptrItemEnd == 0) ){
					p->itemCount = calcItemCount;
					return calcItemCount;
				}
			}

			ptrItemStart = ptrItemEnd;

			if(calcItemCount >= BG_STRINGLIST_MAXITEMCOUNT){
				p->itemCount = calcItemCount;
				return -1;
			}

			/*check for an end of the src string*/
			if( (*ptrItemEnd == 0) ){
				p->itemCount = calcItemCount;
				return calcItemCount;
			}
		}else
		if( *ptrItemEnd == 0){
			p->items[calcItemCount] = ptrItemStart;
			calcItemCount++;
			break;
		}else
			ptrItemEnd++;
	}/*while*/

	p->itemCount = calcItemCount;
	return calcItemCount;
}

int bgStringSplitLineEx(bgStringListEx_typ * p, char separator, char* pLineBuffer, char* pAddrListBuffer, int sizeListBuffer){
unsigned char *ptrItemStart, *ptrItemEnd;
int	calcItemCount;

    p->src = (unsigned char*)pLineBuffer;

    /*if mem data is defined, use it; otherwise, mem shall have been set using a separate call to xxxExMemSet()*/
    if(pAddrListBuffer && sizeListBuffer)
        bgStringListExMemSet(p, pAddrListBuffer, sizeListBuffer);

	p->itemCount = 0;

	ptrItemStart = p->src;
	ptrItemEnd = p->src;

/*process the rest; build list of item pointers*/
	calcItemCount 	= 0;
	while( 1 ){
		if( (*ptrItemEnd == separator) ){
			*ptrItemEnd = 0;
			p->items[calcItemCount] = ptrItemStart;
			ptrItemEnd++;

			calcItemCount++;

			/*check for an additional separtor */
			while( (*ptrItemEnd == separator) ){
				ptrItemEnd++;
				if( (*ptrItemEnd == 0) ){
					p->itemCount = calcItemCount;
					return calcItemCount;
				}
			}

			ptrItemStart = ptrItemEnd;

			if(calcItemCount >= p->itemCountMax){
				p->itemCount = calcItemCount;
				return -1;
			}

			/*check for an end of the src string*/
			if( (*ptrItemEnd == 0) ){
				p->itemCount = calcItemCount;
				return calcItemCount;
			}
		}else
		if( *ptrItemEnd == 0){
			p->items[calcItemCount] = ptrItemStart;
			calcItemCount++;
			break;
		}else
			ptrItemEnd++;
	}/*while*/

	p->itemCount = calcItemCount;
	return calcItemCount;
}

char *bgStringLower(char *s)
{
int i;
char c;

	for(i=0;i<255;i++){

		c = s[i];

		if( !c )
			break;

		if( (c >= 'A') && (c <= 'Z') ){
			s[i] = c - 'A' + 'a';
		}
	}

	return s;
}

char bgCharToLowerCase(char c)
{
char charLowerCase = c;

	if( (c >= 'A') && (c <= 'Z') ){
		charLowerCase = c - 'A' + 'a';
	}

	return charLowerCase;
}

char *bgStringUpper(char *s)
{
int i;
char c;

	for(i=0;i<255;i++){

		c = s[i];

		if( !c )
			break;

		if( (c >= 'a') && (c <= 'z') ){
			s[i] = c - 'a' + 'A';
		}
	}

	return s;
}

int bgStringIsMatch(char *s1, char *s2, int minChrCount)
{
	if( !strcmp(s1, s2) ){
		return 1;
	}else
		return 0;

}

int bgIsNumber_uint(char *s)
{
int i;
char c;

	/*limit execution to 255: don't want cycle time violation due to wrong ptr*/
	for(i=0;i<255;i++){

		c = s[i];

		/*end of valid input string?*/
		if( !c && i)
			return 1;

		/*zero input string?*/
		if( !c && !i)
			return 0;

		/*check if digit or space*/
		if( !bgIsDigit(c) && (c != ' '))
			return 0;
	}

	return 0;
}

int bgIsNumber_int(char *s)
{
int i;
char c;

	/*limit execution to 255: don't want cycle time violation due to wrong ptr*/
	for(i=0;i<255;i++){

		c = s[i];

		/*end of valid input string?*/
		if( !c && i)
			return 1;

		/*zero input string?*/
		if( !c && !i)
			return 0;

		/*check if digit or space*/
		if( !bgIsDigit(c) && (c != ' ') && (c != '-')  && (c != '+'))
			return 0;
	}

	return 0;
}

int bgAsciiToUint(char *src, unsigned int *dst)
{

unsigned int value;

	if( !bgIsNumber_uint(src) )
		return 0;

#ifdef WIN32
	/*TODO!!!*/
	value = 0;
#else
	value = atoi((UDINT)src);
#endif

	*dst = value;

	return 1;
}

int bgAsciiToInt(char *src, unsigned int *dst)
{

unsigned int value;

	if( !bgIsNumber_int(src) )
		return 0;

#ifdef WIN32
	/*TODO!!!*/
	value = 0;
#else
	value = atoi((UDINT)src);
#endif
	*dst = value;

	return 1;
}

int bgStrCopyFromTo(char* src, int srcStartPosition, int srcEndPosition, char* dest)
{
/*
-copy part of the memory from the section of src (from srcStartPosition to srcEndPosition) to dest
-srcEndPosition is not included in the copy (last copied byte position is srcEndPosition-1)
-length of the copied string is (srcEndPosition - srcStartPosition)
Example:
src="01234567890"
srcStartPosition=3
srcEndPosition=7

dest="3456"

return value: number of bytes copied (i.e. length of the dest string)
*/
int size = 0;
int i;

	if( srcEndPosition >= srcStartPosition )
		size = srcEndPosition - srcStartPosition;

	/*do memcopy! end position char is not included in the copy!*/
	for(i=0; i<size; i++)
		dest[i] = src[srcStartPosition + i];

	/*terminate string*/
	dest[size] = 0;

	return size;
}

int bgStrFindEOL(char* src, int startPosition)
{
/*
- search supplied c string "src" (zero terminated!!!) for the eof
- start search at startPosition and look for the first '\n'
- return:
-1 		- EOF (\n) not found
>=0		- EOF position
*/
int position = startPosition;
int i = 0;

	while(1){
		/*end of line?*/
		if( src[position] == '\n' ){
			/*if \r preceeds \n, dec EOL position by 1*/
			if( position && (src[position-1] == '\r') )
				position--;

		 	return position;
		}

 		/*end of string?*/
		if( src[position] == 0 ) return -1;

		/*prevent endless loop*/
		if( ++i >= 4096 ) return -1;

		position++;
	}

	return -1;
}

#endif
/*EOF*/
```
